PROGRAM B_4_2_PRG_Master_ProcessDoor

VAR

	bEventsFlag							: ARRAY [0..100] OF BOOL;
/////////////////////////////////////////////////////////////////////////////////////I O/////////////////////////////////////////////////////////////////////////////////////	
	
	bOpenDoor							: BOOL;
	bCloseDoor							: BOOL;
	bCloseDoorHMI						: BOOL;
	bOpenDoorHMI						: BOOL;
	bDoorClosed							: BOOL;
	tonDoorOpened						: TON;
	bDoorOpened							: BOOL;
	
	bProcessCylinderNotHomed			: BOOL;
	bSlideNestNotHomed					: BOOL;
	
	

	
	
END_VAR

d_ACT_Set_Events_Station_4B();
a_ACT_Ctrl_Station_4B();
b_ACT_IO_B();
c_Manual();

ACTION a_ACT_Ctrl_Station_4B:
/////////////////////////////////////////////////////////////////////////////////////UTILITIES/////////////////////////////////////////////////////////////////////////////////////

/////////////////////////////////////////////////////////////////////////////////////CONDITIONS/////////////////////////////////////////////////////////////////////////////////////
IF stProcessDoor.State <> E_ProcessDoor_State.HOMING THEN
	
	bDoorClosingInitFlag											:= FALSE;

END_IF


IF stProcessDoor.CMD.bAbort THEN
	
	stProcessDoor.State				:= E_ProcessDoor_State.RESET;
	
ELSIF stProcessDoor.CMD.bEndCycle THEN
	
	stProcessDoor.State				:= E_ProcessDoor_State.STOPPING;

END_IF

CASE stProcessDoor.State OF
	
	E_ProcessDoor_State.ABORTED:
	
								IF stProcessDoor.CMD.bEnable THEN
									
									stProcessDoor.State				:= E_ProcessDoor_State.HOMING;
								
								END_IF
								
		E_ProcessDoor_State.HOMING: 
		
								IF bProcessCylinderNotHomed OR bSlideNestNotHomed THEN
									
									bCloseDoor						:= TRUE;
									bOpenDoor						:= FALSE;
									
									IF NOT bDoorClosed AND bCloseDoor THEN
										
										bDoorClosingInitFlag		:= TRUE;
									ELSE bDoorClosingInitFlag		:= FALSE;
									END_IF
									
								ELSE
									
									bCloseDoor						:= FALSE;
									bOpenDoor						:= TRUE;
									
								END_IF
								
								IF bDoorOpened AND NOT (bProcessCylinderNotHomed OR bSlideNestNotHomed) THEN
									
									stProcessDoor.State				:= E_ProcessDoor_State.READY;									
									bOpenDoor						:= FALSE;
																	
								END_IF
	
	
	E_ProcessDoor_State.READY:
	
								IF stProcessDoor.CMD.bExecute AND 	stProcessDoor.CMD.ProcessDoorCMD.OpenDoor	THEN

									stProcessDoor.State				:= E_ProcessDoor_State.OPEN;
									
								ELSIF stProcessDoor.CMD.bExecute AND 	stProcessDoor.CMD.ProcessDoorCMD.CloseDoor	THEN
									
									stProcessDoor.State				:= E_ProcessDoor_State.CLOSE;									
																		
								END_IF
	

	E_ProcessDoor_State.OPEN:
	
								bOpenDoor							:= TRUE;
								
								IF bDoorOpened	THEN
									
									stProcessDoor.State				:= E_ProcessDoor_State.DONE;
								
								END_IF
								
	E_ProcessDoor_State.CLOSE:
	
								bCloseDoor							:= TRUE;
								
								IF bDoorClosed THEN
									
									stProcessDoor.State				:= E_ProcessDoor_State.DONE;
								
								END_IF
								
	E_ProcessDoor_State.DONE:
	
	
								IF stProcessDoor.CMD.bAcknowledge THEN
									
									stProcessDoor.CMD.bAcknowledge	:= FALSE;
									stProcessDoor.State				:= E_ProcessDoor_State.RESET;
								
								END_IF
	
	
	E_ProcessDoor_State.RESET:	
	
								bOpenDoor							:= FALSE;
								bCloseDoor							:= FALSE;
								
								IF NOT stProcessDoor.CMD.bAbort AND NOT stProcessDoor.CMD.bEndCycle THEN
									
									stProcessDoor.State				:= E_ProcessDoor_State.READY;
									
								ELSE stProcessDoor.State			:= E_ProcessDoor_State.ABORTED;
								END_IF
	
					
	E_ProcessDoor_State.STOPPING:					
									
								bOpenDoor							:= TRUE;
									
								IF bDoorOpened THEN
									
									bOpenDoor						:= FALSE;
									stProcessDoor.State				:= E_ProcessDoor_State.RESET;
								
								END_IF
								
							
														
									

ELSE stProcessDoor.State		:= E_ProcessDoor_State.ABORTED;
	
END_CASE
/////////////////////////////////////////////////////////////////////////////////////STATUS/////////////////////////////////////////////////////////////////////////////////////

stProcessDoor.Status.bBusy			:= 	stProcessDoor.State	= E_ProcessDoor_State.CLOSE OR
										stProcessDoor.State	= E_ProcessDoor_State.OPEN OR 
										stProcessDoor.State	= E_ProcessDoor_State.STOPPING;
								
stProcessDoor.Status.bDone			:=	stProcessDoor.State	= E_ProcessDoor_State.DONE;

stProcessDoor.Status.bReady			:= 	stProcessDoor.State	= E_ProcessDoor_State.READY;

stProcessDoor.Status.bStopped		:= 	NOT stProcessDoor.Status.bBusy;
END_ACTION

ACTION b_ACT_IO_B:
tonDoorOpened( IN := NOT bDoorClosed, PT := stTimers.tDoorOpenedSignal);


bDoorClosed								:= dw_T05_EL1918.iProcessDoorClosed1 AND dw_T05_EL1918.iProcessDoorClosed2 AND dw_T05_EL1918.iProcessDoorFB;
bDoorOpened								:= tonDoorOpened.Q; 
bProcessDoorClosed						:= bDoorClosed;

bDoorOpenedFlag							:= bDoorOpened;

dw_T09_EL2809.qOpenProcessDoor			:= bOpenDoor OR bOpenDoorHMI OR stStationEvents[4].aEvents[0].bEventTimer.Q;//OR bOpenDoorCycleFault;	
dw_T09_EL2809.qCloseProcessDoor			:= bCloseDoor OR bCloseDoorHMI;

bProcessCylinderNotHomed				:= NOT stTwinSAFE.qProcessCylinderRetracted;
bSlideNestNotHomed						:= NOT dw_T08_EL1809.iSlideNestRetracted;
END_ACTION

ACTION c_Manual:


IF bProcessDoor_Down AND stTwinSAFE.qTwoHandsSafe THEN
	
	bCloseDoorHMI					:= TRUE;
	bProcessDoor_Down				:= FALSE;
	
ELSIF bDoorClosed  OR NOT stMachineStatus.bManualMode THEN

	 bCloseDoorHMI					:= FALSE;
	 bProcessDoor_Down				:= FALSE;

END_IF

IF bProcessDoor_UP THEN
	
	bOpenDoorHMI					:= TRUE;
	
	
ELSIF bDoorOpened OR  NOT stMachineStatus.bManualMode THEN

	bOpenDoorHMI					:= FALSE;	 
	
END_IF
END_ACTION

ACTION d_ACT_Set_Events_Station_4B:
//IMMEDIATE FAULTS

stStationEvents[4].aEvents[0].bEventTimer( IN :=  (bCloseDoor OR bCloseDoorHMI) AND NOT bDoorClosed, PT := T#2S);
stStationEvents[4].aEvents[0].bFault						:= TRUE;
stStationEvents[4].aEvents[0].bEventFlag					:= stStationEvents[4].aEvents[0].bEventTimer.Q;
stStationEvents[4].aEvents[0].bEventText					:= 'Process Door extend timeout';
stStationEvents[4].aEvents[0].sSolution						:= 'Check cylinder, neumatic connections and sensors';

stStationEvents[4].aEvents[1].bEventTimer( IN :=  (bOpenDoor OR bOpenDoorHMI) AND NOT bDoorOpened, PT := T#2S);
stStationEvents[4].aEvents[1].bFault						:= TRUE;
stStationEvents[4].aEvents[1].bEventFlag					:= stStationEvents[4].aEvents[1].bEventTimer.Q;
stStationEvents[4].aEvents[1].bEventText					:= 'Process Door Retract timeout';
stStationEvents[4].aEvents[1].sSolution						:= 'Check cylinder, neumatic connections and sensors';





//CYCLE STOP REQUEST

(*stStationEvents[4].aEvents[2].bCycleStopRequest			:= TRUE;
stStationEvents[4].aEvents[2].bEventFlag					:= bEventsFlag[2];
stStationEvents[4].aEvents[2].bEventText					:= 'ST1 EVENT 7';*)
END_ACTION

END_PROGRAM

(* stored: Version 1.1.0.1, ProductVersion 3.1.4026.18
   POU B_4_2_PRG_Master_ProcessDoor: Id {53a11cee-2388-4375-a004-26a2c48b086a}, SpecialFunc None
   Action a_ACT_Ctrl_Station_4B: Id {08b1d871-01b9-45fa-bb18-30d558502fc6}
   Action b_ACT_IO_B: Id {7a24ac88-21cc-4219-af73-2aba76419ebf}
   Action c_Manual: Id {af74f668-26ed-493a-861d-9af0f131bf72}
   Action d_ACT_Set_Events_Station_4B: Id {6917e64e-8f14-430a-8afe-2820b830fd4d} *)
